// TwinCAT 3 PLC project PLC1
// ProgramVersion: 3.1.4023.0
// libraries:
//   Tc2_Standard, * (Beckhoff Automation GmbH)
//   Tc2_System, * (Beckhoff Automation GmbH)
//   Tc3_Module, * (Beckhoff Automation GmbH)
// project tree:
//   GVLs/ GVL1.TcGVL
//   / PlcTask.TcTTO
//   POUs/ MAIN.TcPOU
// real-time tasks:
//   TASK PlcTask: cycle T#10ms, priority 20, ADS port 341

CONFIGURATION PLC1
    RESOURCE PLC ON TwinCAT3
        TASK PlcTask(INTERVAL := T#10ms, PRIORITY := 20);
        PROGRAM MAIN WITH PlcTask : MAIN;
    END_RESOURCE
END_CONFIGURATION

// ---- GVLs/GVL1.TcGVL
{attribute 'qualified_only'}
VAR_GLOBAL
	Switch:BOOL;
	Lamp:bool;
END_VAR

// ---- POUs/MAIN.TcPOU
PROGRAM MAIN
VAR
	T1: TON;
END_VAR

T1(IN:=GVL1.Switch , PT:=T#5s , Q=>GVL1.Lamp );

END_PROGRAM
